# EPICS substitutions: hugo/source/db/Beckhoff_1XXX/ecmcEL1144.substitutions
# binary inputs
file "ecmc_binaryInput-chX.template"{
  pattern {CH_ID}
          {01   }
          {02   }
          {03   }
          {04   }
}
